// TIA Portal V17 export
// export: Created 2025-03-07T09:18:24.1596422Z, ExportSetting WithDefaults, DisplayName Totally Integrated Automation Portal, DisplayVersion V17 Update 8, DisplayName TIA Portal Openness, DisplayVersion V17 Update 8, DisplayName TIA Portal Version Control Interface, DisplayVersion V17, DisplayName SINAMICS Startdrive Advanced, DisplayVersion V17 SP2, DisplayName SINAMICS Startdrive G110M, G120, G120C, G120D, G120P, G115D, DisplayVersion V17 SP2, DisplayName SINAMICS Startdrive G130, G150, S120, S150, SINAMICS MV, S210, DisplayVersion V17 SP2, DisplayName STEP 7 Professional, DisplayVersion V17 Update 8, DisplayName SINUMERIK ONE STEP 7 Toolbox, DisplayVersion V17 Update 12, DisplayName SINUMERIK 840D sl STEP 7 Toolbox, DisplayVersion V17 Update 12, DisplayName STEP 7 Safety, DisplayVersion V17 Update 6, DisplayName WinCC Advanced, DisplayVersion V17 Update 8
DATA_BLOCK "DB1451_MAIN_COOLING_SYSTEM"   // DB1451
{ S7_Optimized_Access := 'FALSE'; DB_Accessible_From_OPC_UA := 'FALSE' }
VERSION : 0.1
// stored: AutoNumber false, DBAccessibleFromOPCUA false, DBAccessibleFromWebserver true, IsOnlyStoredInLoadMemory false, IsWriteProtectedInAS false
   VAR
      COOLING_INPUT_SENSOR : Struct
         COOLING_FLOW_SENSOR_VALUE : Real;   // MACHINE COOLING INPUT FLOW SENSOR VALUE
         COOLING_TEMP_SENSOR_VALUE : Real;   // MACHINE COOLING INPUT TEMP SENSOR VALUE
         COOLING_FLOW_LOW_WARNING_VALUE : Real;   // MACHINE COOLING INPUT FLOW LOW WARNING VALUE
         COOLING_FLOW_HIGH_WARNING_VALUE : Real;   // MACHINE COOLING INPUT FLOW HIGH WARNING VALUE
         COOLING_FLOW_LOW_ALARM_VALUE : Real;   // MACHINE COOLING INPUT FLOW LOW ALARM VALUE
         COOLING_FLOW_HIGH_ALARM_VALUE : Real;   // MACHINE COOLING INPUT FLOW HIGH ALARM VALUE
         COOLING_TEMP_LOW_WARNING_VALUE : Real;   // MACHINE COOLING INPUT TEMP LOW WARNING VALUE
         COOLING_TEMP_HIGH_WARNING_VALUE : Real;   // MACHINE COOLING INPUT TEMP HIGH WARNING VALUE
         COOLING_TEMP_LOW_ALARM_VALUE : Real;   // MACHINE COOLING INPUT TEMP LOW ALARM VALUE
         "COOLING_TEMP_HIGH ALARM_VALUE" : Real;   // MACHINE COOLING INPUT TEMP HIGH ALARM VALUE
         WARNINGS : Struct
            COOLING_FLOW_LOW_WARNING : Bool;   // MACHINE COOLING INPUT FLOW LOW WARNING
            COOLING_FLOW_HIGH_WARNING : Bool;   // MACHINE COOLING INPUT FLOW HIGH WARNING
            COOLING_TEMP_LOW_WARNING : Bool;   // MACHINE COOLING INPUT TEMPERATURE LOW WARNING
            COOLING_TEMP_HIGH_WARNING : Bool;   // MACHINE COOLING INPUT TEMPERATURE HIGH WARNINGS
         END_STRUCT;
         ALARMS : Struct
            COOLING_FLOW_LOW_ALARM : Bool;   // MACHINE COOLING FLOW LOW ALARM
            COOLING_FLOW_HIGH_ALARM : Bool;   // MACHINE COOLING FLOW HIGH ALARM
            COOLING_TEMP_LOW_ALARM : Bool;   // MACHINE COOLING TEMPERATURE LOW ALARM
            COOLING_TEMP_HIGH_ALARM : Bool;   // MACHINE COOLING TEMPERATURE HIGH ALARM
            COOLING_FLOW_SETPOINT_ALARM : Bool;   // MACHINE COOLING FLOW SETPOINT ALARM
            COOLING_TEMP_SETPOINT_ALARM : Bool;   // MACHINE COOLING TEMPERATURE SETPOINT ALARM
         END_STRUCT;
      END_STRUCT;
      COOLING_OUTPUT_SENSOR : Struct
         COOLING_FLOW_SENSOR_VALUE : Real;   // MACHINE COOLING OUTPUT FLOW SENSOR VALUE
         COOLING_TEMP_SENSOR_VALUE : Real;   // MACHINE COOLING OUTPUT TEMP SENSOR VALUE
         COOLING_FLOW_LOW_WARNING_VALUE : Real;   // MACHINE COOLING INPUT OUTPUT LOW WARNING VALUE
         COOLING_FLOW_HIGH_WARNING_VALUE : Real;   // MACHINE COOLING OUTPUT FLOW HIGH WARNING VALUE
         COOLING_FLOW_LOW_ALARM_VALUE : Real;   // MACHINE COOLING OUTPUT FLOW LOW ALARM VALUE
         COOLING_FLOW_HIGH_ALARM_VALUE : Real;   // MACHINE COOLING OUTPUT FLOW HIGH ALARM VALUE
         COOLING_TEMP_LOW_WARNING_VALUE : Real;   // MACHINE COOLING OUTPUT TEMP LOW WARNING VALUE
         COOLING_TEMP_HIGH_WARNING_VALUE : Real;   // MACHINE COOLING OUTPUT TEMP HIGH WARNING VALUE
         COOLING_TEMP_LOW_ALARM_VALUE : Real;   // MACHINE COOLING OUTPUT TEMP LOW ALARM VALUE
         "COOLING_TEMP_HIGH ALARM_VALUE" : Real;   // MACHINE COOLING OUTPUT TEMP HIGH ALARM VALUE
         WARNINGS : Struct
            COOLING_FLOW_LOW_WARNING : Bool;   // MACHINE COOLING OUTPUT FLOW LOW WARNING
            COOLING_FLOW_HIGH_WARNING : Bool;   // MACHINE COOLING OUTPUT FLOW HIGH WARNING
            COOLING_TEMP_LOW_WARNING : Bool;   // MACHINE COOLING OUTPUT TEMPERATURE LOW WARNING
            COOLING_TEMP_HIGH_WARNING : Bool;   // MACHINE COOLING OUTPUT TEMPERATURE HIGH WARNINGS
         END_STRUCT;
         ALARMS : Struct
            COOLING_FLOW_LOW_ALARM : Bool;   // MACHINE COOLING OUTPUT FLOW LOW ALARM
            COOLING_FLOW_HIGH_ALARM : Bool;   // MACHINE COOLING OUTPUT FLOW HIGH ALARM
            COOLING_TEMP_LOW_ALARM : Bool;   // MACHINE COOLING OUTPUT TEMPERATURE LOW ALARM
            COOLING_TEMP_HIGH_ALARM : Bool;   // MACHINE COOLING OUTPUT TEMPERATURE HIGH ALARM
            COOLING_FLOW_SETPOINT_ALARM : Bool;   // MACHINE COOLING OUTPUT FLOW SETPOINT ALARM
            COOLING_TEMP_SETPOINT_ALARM : Bool;   // MACHINE COOLING OUTPUT TEMPERATURE SETPOINT ALARM
         END_STRUCT;
      END_STRUCT;
   END_VAR
BEGIN
END_DATA_BLOCK
